TYPE ST_ProBoxSafetyOutputsLowLift :
STRUCT
	FeedBackK1				: BOOL; // First feedback signal for LowLift 
	FeedBackK2				: BOOL; // Second feedback signal for Lowlift 	
	ContactorOn             : BOOL; //Send button to safety
	ContactorOff            : BOOL; //Send button to safety
	ResetSafetyNeeded       : BOOL; //Indication I/O output 
	ErrorAck                : BOOL; //Error acknowledgement sent to safety
	TransportActive			: bool;	//Transport active
END_STRUCT
END_TYPE

(* stored: Version 1.1.0.1, ProductVersion 3.1.4024.4
   DUT ST_ProBoxSafetyOutputsLowLift: Id {7304dca1-7a5b-4c4f-941d-44bfab5d7945} *)
